// Mitsubishi GX Works2 project: BookEX6_17 Output   PLC: Q13UDV

// global labels: Global
VAR_GLOBAL
  bVar0 AT M5000 : BOOL;
  abArray0 AT M5010 : ARRAY [0..49] OF BOOL;
  sStr0 AT D5000 : STRING[199];
  sStr1 AT D5100 : STRING[199];
  sStr2 AT D5200 : STRING[199];
  sStr3 AT D5300 : STRING[199];
  sStr4 AT D5400 : STRING[199];
  sStr5 AT D5500 : STRING[199];
  sStr6 AT D5600 : STRING[199];
  sStr7 AT D5700 : STRING[199];
  sStr8 AT D5800 : STRING[199];
  sStr9 AT D5900 : STRING[199];
  iVar0 AT D4500 : INT;
  iVar1 AT D4501 : INT;
  iVar2 AT D4502 : INT;
  iVar3 AT D4503 : INT;
  iVar4 AT D4504 : INT;
  iVar5 AT D4505 : INT;
  iVar6 AT D4506 : INT;
  iVar7 AT D4507 : INT;
  iVar8 AT D4508 : INT;
  iVar9 AT D4509 : INT;
  dVar0 AT D4510 : DINT;
  dVar1 AT D4512 : DINT;
  dVar2 AT D4514 : DINT;
  dVar3 AT D4516 : DINT;
  dVar4 AT D4518 : DINT;
  dVar5 AT D4520 : DINT;
  dVar6 AT D4522 : DINT;
  dVar7 AT D4524 : DINT;
  dVar8 AT D4526 : DINT;
  dVar9 AT D4528 : DINT;
  wVar0 AT D4530 : WORD;
  wVar1 AT D4531 : WORD;
  wVar2 AT D4532 : WORD;
  wVar3 AT D4533 : WORD;
  wVar4 AT D4534 : WORD;
  wVar5 AT D4535 : WORD;
  wVar6 AT D4536 : WORD;
  wVar7 AT D4537 : WORD;
  wVar8 AT D4538 : WORD;
  wVar9 AT D4539 : WORD;
  dwVar0 AT D4540 : DWORD;
  dwVar1 AT D4542 : DWORD;
  dwVar2 AT D4544 : DWORD;
  dwVar3 AT D4546 : DWORD;
  dwVar4 AT D4548 : DWORD;
  dwVar5 AT D4550 : DWORD;
  dwVar6 AT D4552 : DWORD;
  dwVar7 AT D4554 : DWORD;
  dwVar8 AT D4556 : DWORD;
  dwVar9 AT D4558 : DWORD;
  fsVar0 AT D4560 : REAL;
  fsVar1 AT D4562 : REAL;
  fsVar2 AT D4564 : REAL;
  fsVar3 AT D4566 : REAL;
  fsVar4 AT D4568 : REAL;
  fsVar5 AT D4570 : REAL;
  fsVar6 AT D4572 : REAL;
  fsVar7 AT D4574 : REAL;
  fsVar8 AT D4576 : REAL;
  fsVar9 AT D4578 : REAL;
  fdVar0 AT D4580 : LREAL;
  tTime0 AT D4620 : TIME;
  tTime1 AT D4622 : TIME;
  tTime2 AT D4624 : TIME;
  tTime3 AT D4626 : TIME;
  tTime4 AT D4628 : TIME;
  tTime5 AT D4630 : TIME;
  tTime6 AT D4632 : TIME;
  tTime7 AT D4634 : TIME;
  tTime8 AT D4636 : TIME;
  tTime9 AT D4638 : TIME;
  tTime10 AT D4640 : TIME;
  bVar1 AT M5001 : BOOL;
  bVar2 AT M5002 : BOOL;
  bVar3 AT M5003 : BOOL;
  bVar4 AT M5004 : BOOL;
  bVar5 AT M5005 : BOOL;
  bVar6 AT M5006 : BOOL;
  bVar7 AT M5007 : BOOL;
  bVar8 AT M5008 : BOOL;
  bVar9 AT M5009 : BOOL;
  abArray1 AT M5060 : ARRAY [0..49] OF BOOL;
  abArray2 AT M5110 : ARRAY [0..49] OF BOOL;
  abArray3 AT M5160 : ARRAY [0..49] OF BOOL;
  abArray4 AT M5210 : ARRAY [0..49] OF BOOL;
  abArray5 AT M5260 : ARRAY [0..49] OF BOOL;
  abArray6 AT M5310 : ARRAY [0..49] OF BOOL;
  abArray7 AT M5360 : ARRAY [0..49] OF BOOL;
  abArray8 AT M5410 : ARRAY [0..49] OF BOOL;
  abArray9 AT M5460 : ARRAY [0..49] OF BOOL;
  fdVar1 AT D4584 : LREAL;
  fdVar2 AT D4588 : LREAL;
  fdVar3 AT D4592 : LREAL;
  fdVar4 AT D4596 : LREAL;
  fdVar5 AT D4600 : LREAL;
  fdVar6 AT D4604 : LREAL;
  fdVar7 AT D4608 : LREAL;
  fdVar8 AT D4612 : LREAL;
  fdVar9 AT D4616 : LREAL;
  aSendData1 AT D100 : ARRAY [0..9] OF INT;
  aiTxData AT D4000 : ARRAY [0..99] OF INT;
  aiRxData AT D4100 : ARRAY [0..99] OF INT;
  iOpenOK AT D3900 : INT;
  iOpenERR AT D3901 : INT;
  iSendOK AT D3902 : INT;
  iSendERR AT D3903 : INT;
  iCloseOK AT D3906 : INT;
  iCloseERR AT D3907 : INT;
  iRecvOK AT D3904 : INT;
  iRecvERR AT D3905 : INT;
  aiTxData2 AT D4200 : ARRAY [0..99] OF INT;
  aiRxData2 AT D4300 : ARRAY [0..99] OF INT;
  iOpenOK2 AT D3908 : INT;
  iOpenERR2 AT D3909 : INT;
  iSendOK2 AT D3910 : INT;
  iSendERR2 AT D3911 : INT;
  iRecvOK2 AT D3912 : INT;
  iRecvERR2 AT D3913 : INT;
  iCloseOK2 AT D3914 : INT;
  iCloseERR2 AT D3915 : INT;
  iEOpenComp AT D3916 : INT;
  iEOpenReq AT D3917 : INT;
  iERecvFlag AT D3918 : INT;
  iOpenCode AT D3919 : INT;
  iSendCode AT D3920 : INT;
  iRecvCode AT D3921 : INT;
  iCloseCode AT D3922 : INT;
  iOpenCode2 AT D3923 : INT;
  iSendCode2 AT D3924 : INT;
  iRecvCode2 AT D3925 : INT;
  iCloseCode2 AT D3926 : INT;
  aRecvData1 AT D110 : ARRAY [0..9] OF INT;
  aSendData2 AT D120 : ARRAY [0..9] OF INT;
  aRecvData2 AT D130 : ARRAY [0..9] OF INT;
END_VAR
// user libraries (not included): HMI

FUNCTION_BLOCK Flicker
VAR_INPUT
  t_Duty : TIME;
END_VAR
VAR_OUTPUT
  b_Lamp1 : BOOL;
  b_Lamp2 : BOOL;
END_VAR
VAR
  iInterval : INT;
END_VAR
;
iInterval := TIME_TO_INT(t_Duty) / 100;
OUT_T(NOT TS1, TC0, iInterval);
OUT_T(TS0, TC1, iInterval);
b_Lamp1 := TS0;
b_Lamp2 :=  NOT TS0;
END_FUNCTION_BLOCK

PROGRAM ExDELTA
VAR
  HMI05_1 : HMI05;
END_VAR
(* structured ladder/FBD written out as ST: instructions are called as NAME(EN, inputs, outputs); _pN, _eN, _tN stand for wires *)
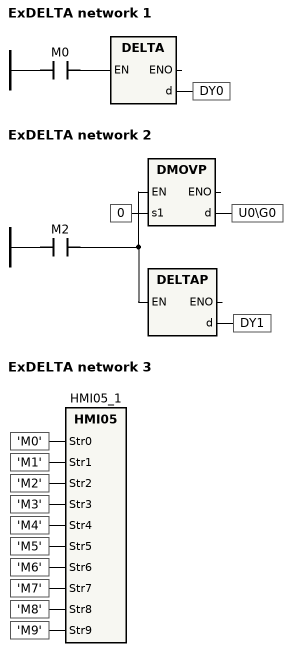
(* network 1 *)
DELTA(M0, DY0);
(* network 2 *)
DMOVP(M2, 0, U0\G0);
DELTAP(M2, DY1);
(* network 3 *)
HMI05_1(Str0 := 'M0', Str1 := 'M1', Str2 := 'M2', Str3 := 'M3', Str4 := 'M4', Str5 := 'M5', Str6 := 'M6', Str7 := 'M7', Str8 := 'M8', Str9 := 'M9');
END_PROGRAM

PROGRAM ExFF
VAR
  HMI05_1 : HMI05;
END_VAR
(* structured ladder/FBD written out as ST: instructions are called as NAME(EN, inputs, outputs); _pN, _eN, _tN stand for wires *)
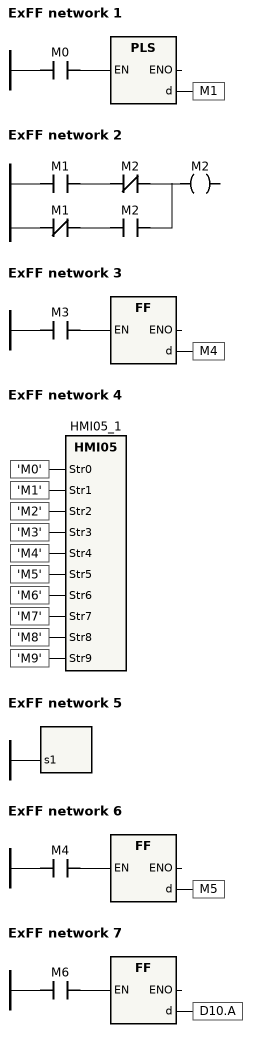
(* network 1 *)
PLS(M0, M1);
(* network 2 *)
M2 := (M1 AND NOT M2) OR (NOT M1 AND M2);
(* network 3 *)
FF(M3, M4);
(* network 4 *)
HMI05_1(Str0 := 'M0', Str1 := 'M1', Str2 := 'M2', Str3 := 'M3', Str4 := 'M4', Str5 := 'M5', Str6 := 'M6', Str7 := 'M7', Str8 := 'M8', Str9 := 'M9');
(* network 5 *)
(* element kind 10  <- TRUE *)
(* network 6 *)
FF(M4, M5);
(* network 7 *)
FF(M6, D10.A);
END_PROGRAM

PROGRAM ExFlicker
VAR
  HMI05_1 : HMI05;
  Flicker_1 : Flicker;
END_VAR
(* structured ladder/FBD written out as ST: instructions are called as NAME(EN, inputs, outputs); _pN, _eN, _tN stand for wires *)
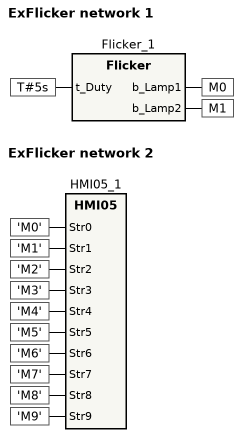
(* network 1 *)
Flicker_1(t_Duty := T#5s, b_Lamp1 => M0, b_Lamp2 => M1);
(* network 2 *)
HMI05_1(Str0 := 'M0', Str1 := 'M1', Str2 := 'M2', Str3 := 'M3', Str4 := 'M4', Str5 := 'M5', Str6 := 'M6', Str7 := 'M7', Str8 := 'M8', Str9 := 'M9');
END_PROGRAM

PROGRAM ExOUT
VAR
  HMI05_1 : HMI05;
END_VAR
(* structured ladder/FBD written out as ST: instructions are called as NAME(EN, inputs, outputs); _pN, _eN, _tN stand for wires *)
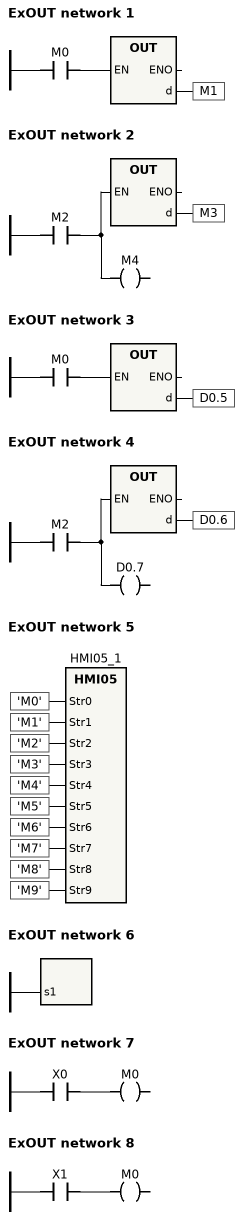
(* network 1 *)
OUT(M0, M1);
(* network 2 *)
OUT(M2, M3);
M4 := M2;
(* network 3 *)
OUT(M0, D0.5);
(* network 4 *)
OUT(M2, D0.6);
D0.7 := M2;
(* network 5 *)
HMI05_1(Str0 := 'M0', Str1 := 'M1', Str2 := 'M2', Str3 := 'M3', Str4 := 'M4', Str5 := 'M5', Str6 := 'M6', Str7 := 'M7', Str8 := 'M8', Str9 := 'M9');
(* network 6 *)
(* element kind 10  <- TRUE *)
(* network 7 *)
M0 := X0;
(* network 8 *)
M0 := X1;
END_PROGRAM

PROGRAM ExOut_C
VAR
  HMI05_1 : HMI05;
END_VAR
(* structured ladder/FBD written out as ST: instructions are called as NAME(EN, inputs, outputs); _pN, _eN, _tN stand for wires *)
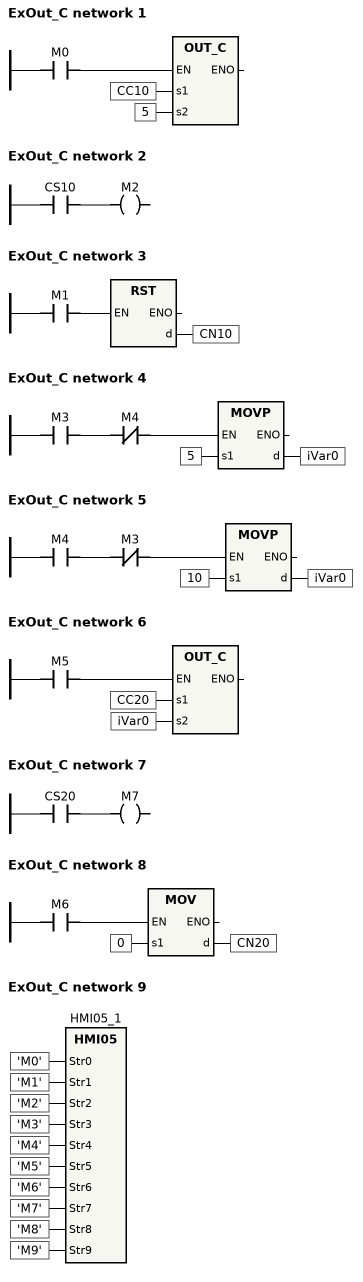
(* network 1 *)
OUT_C(M0, CC10, 5);
(* network 2 *)
M2 := CS10;
(* network 3 *)
RST(M1, CN10);
(* network 4 *)
MOVP(M3 AND NOT M4, 5, iVar0);
(* network 5 *)
MOVP(M4 AND NOT M3, 10, iVar0);
(* network 6 *)
OUT_C(M5, CC20, iVar0);
(* network 7 *)
M7 := CS20;
(* network 8 *)
MOV(M6, 0, CN20);
(* network 9 *)
HMI05_1(Str0 := 'M0', Str1 := 'M1', Str2 := 'M2', Str3 := 'M3', Str4 := 'M4', Str5 := 'M5', Str6 := 'M6', Str7 := 'M7', Str8 := 'M8', Str9 := 'M9');
END_PROGRAM

PROGRAM ExOut_T
VAR
  HMI05_1 : HMI05;
END_VAR
(* structured ladder/FBD written out as ST: instructions are called as NAME(EN, inputs, outputs); _pN, _eN, _tN stand for wires *)
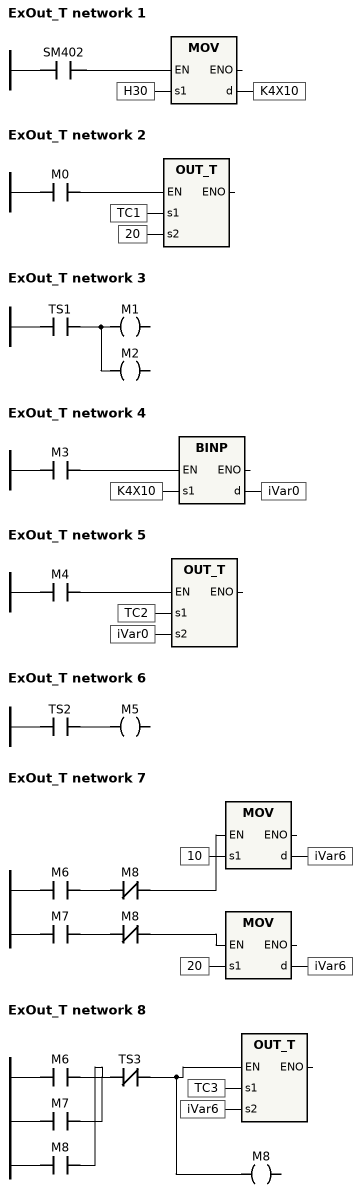
(* network 1 *)
MOV(SM402, H30, K4X10);
(* network 2 *)
OUT_T(M0, TC1, 20);
(* network 3 *)
M1 := TS1;
M2 := TS1;
(* network 4 *)
BINP(M3, K4X10, iVar0);
(* network 5 *)
OUT_T(M4, TC2, iVar0);
(* network 6 *)
M5 := TS2;
(* network 7 *)
MOV(M6 AND NOT M8, 10, iVar6);
MOV(M7 AND NOT M8, 20, iVar6);
(* network 8 *)
_p1 := (M6 OR M7 OR M8) AND NOT TS3;
M8 := _p1;
OUT_T(_p1, TC3, iVar6);
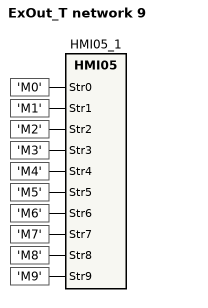
(* network 9 *)
HMI05_1(Str0 := 'M0', Str1 := 'M1', Str2 := 'M2', Str3 := 'M3', Str4 := 'M4', Str5 := 'M5', Str6 := 'M6', Str7 := 'M7', Str8 := 'M8', Str9 := 'M9');
END_PROGRAM

PROGRAM ExOut_T2
VAR
  HMI05_1 : HMI05;
END_VAR
(* structured ladder/FBD written out as ST: instructions are called as NAME(EN, inputs, outputs); _pN, _eN, _tN stand for wires *)
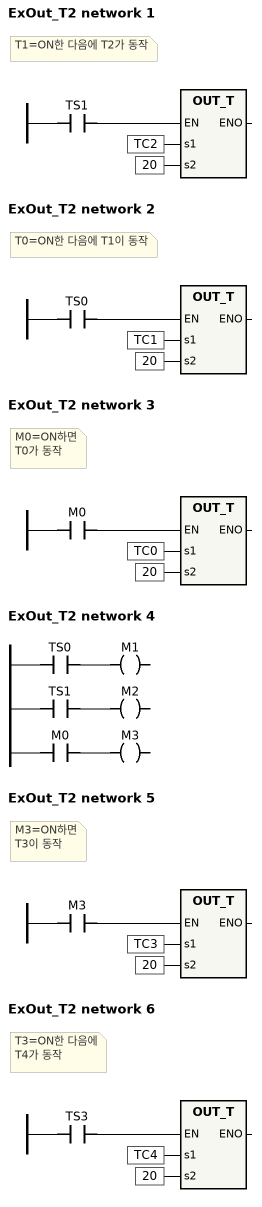
(* network 1 *)
(* T1=ON한 다음에 T2가 동작 *)
OUT_T(TS1, TC2, 20);
(* network 2 *)
(* T0=ON한 다음에 T1이 동작 *)
OUT_T(TS0, TC1, 20);
(* network 3 *)
(* M0=ON하면  / T0가 동작 *)
OUT_T(M0, TC0, 20);
(* network 4 *)
M1 := TS0;
M2 := TS1;
M3 := M0;
(* network 5 *)
(* M3=ON하면  / T3이 동작 *)
OUT_T(M3, TC3, 20);
(* network 6 *)
(* T3=ON한 다음에  / T4가 동작 *)
OUT_T(TS3, TC4, 20);
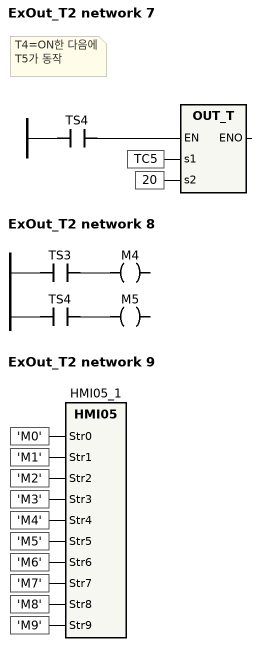
(* network 7 *)
(* T4=ON한 다음에  / T5가 동작 *)
OUT_T(TS4, TC5, 20);
(* network 8 *)
M4 := TS3;
M5 := TS4;
(* network 9 *)
HMI05_1(Str0 := 'M0', Str1 := 'M1', Str2 := 'M2', Str3 := 'M3', Str4 := 'M4', Str5 := 'M5', Str6 := 'M6', Str7 := 'M7', Str8 := 'M8', Str9 := 'M9');
END_PROGRAM

PROGRAM ExPLF
VAR
  HMI05_1 : HMI05;
END_VAR
(* structured ladder/FBD written out as ST: instructions are called as NAME(EN, inputs, outputs); _pN, _eN, _tN stand for wires *)
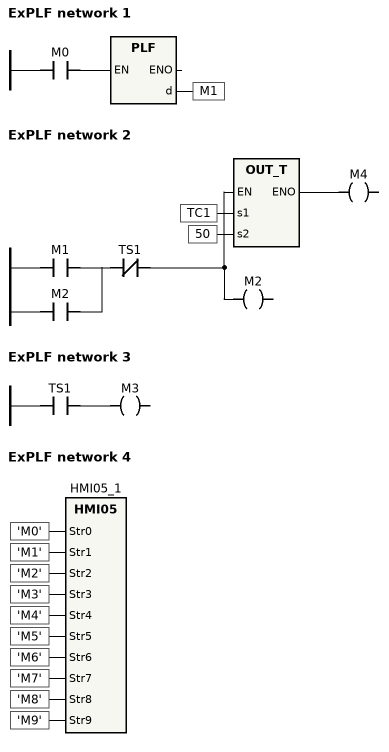
(* network 1 *)
PLF(M0, M1);
(* network 2 *)
_p1 := (M1 OR M2) AND NOT TS1;
_e2 := OUT_T(_p1, TC1, 50);
M4 := _e2;
M2 := _p1;
(* network 3 *)
M3 := TS1;
(* network 4 *)
HMI05_1(Str0 := 'M0', Str1 := 'M1', Str2 := 'M2', Str3 := 'M3', Str4 := 'M4', Str5 := 'M5', Str6 := 'M6', Str7 := 'M7', Str8 := 'M8', Str9 := 'M9');
END_PROGRAM

PROGRAM ExPLS
VAR
  HMI05_1 : HMI05;
END_VAR
(* structured ladder/FBD written out as ST: instructions are called as NAME(EN, inputs, outputs); _pN, _eN, _tN stand for wires *)
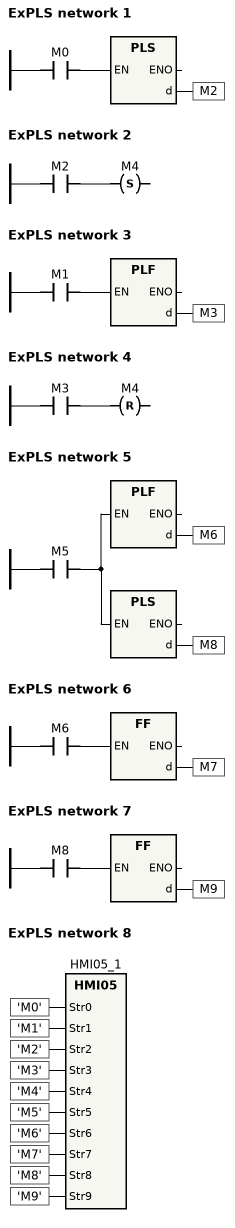
(* network 1 *)
PLS(M0, M2);
(* network 2 *)
SET(M2, M4);
(* network 3 *)
PLF(M1, M3);
(* network 4 *)
RST(M3, M4);
(* network 5 *)
PLF(M5, M6);
PLS(M5, M8);
(* network 6 *)
FF(M6, M7);
(* network 7 *)
FF(M8, M9);
(* network 8 *)
HMI05_1(Str0 := 'M0', Str1 := 'M1', Str2 := 'M2', Str3 := 'M3', Str4 := 'M4', Str5 := 'M5', Str6 := 'M6', Str7 := 'M7', Str8 := 'M8', Str9 := 'M9');
END_PROGRAM

PROGRAM ExPowerOn
VAR
  bPowerFail : BOOL;
  TON_1 : TON;
  TON_2 : TON;
  bOff : BOOL;
  bOn : BOOL;
  TON_3 : TON;
  HMI05_1 : HMI05;
END_VAR
(* structured ladder/FBD written out as ST: instructions are called as NAME(EN, inputs, outputs); _pN, _eN, _tN stand for wires *)
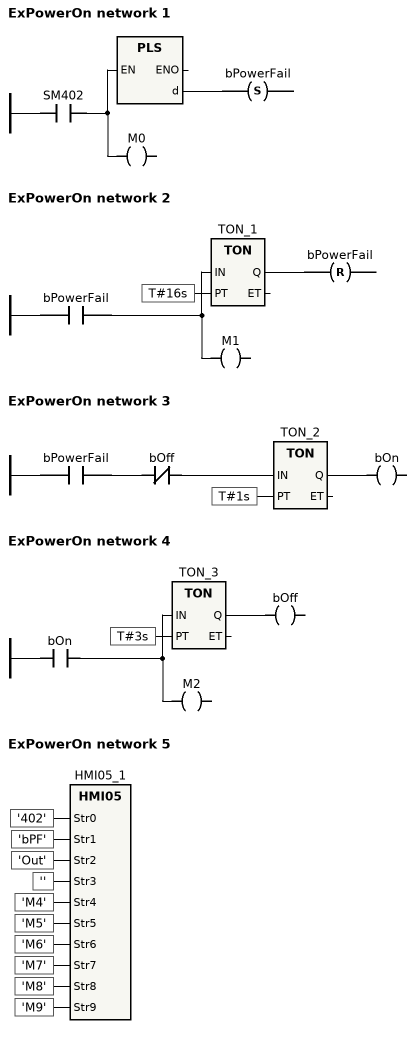
(* network 1 *)
PLS(SM402, _t1);
SET(_t1, bPowerFail);
M0 := SM402;
(* network 2 *)
TON_1(IN := bPowerFail, PT := T#16s);
RST(TON_1.Q, bPowerFail);
M1 := bPowerFail;
(* network 3 *)
TON_2(IN := bPowerFail AND NOT bOff, PT := T#1s);
bOn := TON_2.Q;
(* network 4 *)
TON_3(IN := bOn, PT := T#3s);
bOff := TON_3.Q;
M2 := bOn;
(* network 5 *)
HMI05_1(Str0 := '402', Str1 := 'bPF', Str2 := 'Out', Str3 := '', Str4 := 'M4', Str5 := 'M5', Str6 := 'M6', Str7 := 'M7', Str8 := 'M8', Str9 := 'M9');
END_PROGRAM

PROGRAM ExPowerOn2
VAR
  bPowerFail : BOOL;
  TON_1 : TON;
  TON_2 : TON;
  bOff : BOOL;
  bOn : BOOL;
  TON_3 : TON;
  HMI05_1 : HMI05;
END_VAR
(* structured ladder/FBD written out as ST: instructions are called as NAME(EN, inputs, outputs); _pN, _eN, _tN stand for wires *)
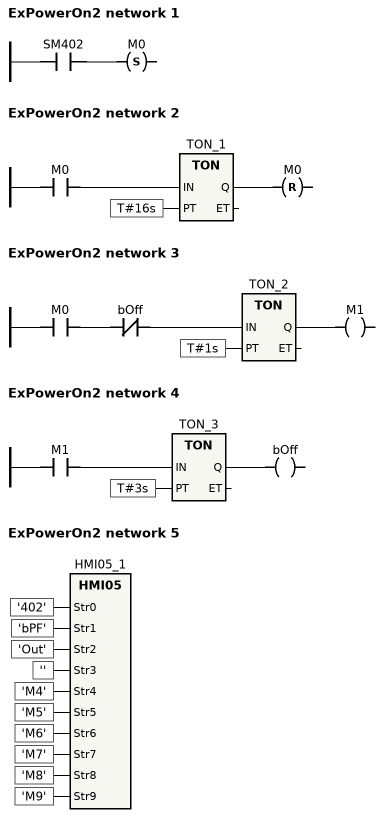
(* network 1 *)
SET(SM402, M0);
(* network 2 *)
TON_1(IN := M0, PT := T#16s);
RST(TON_1.Q, M0);
(* network 3 *)
TON_2(IN := M0 AND NOT bOff, PT := T#1s);
M1 := TON_2.Q;
(* network 4 *)
TON_3(IN := M1, PT := T#3s);
bOff := TON_3.Q;
(* network 5 *)
HMI05_1(Str0 := '402', Str1 := 'bPF', Str2 := 'Out', Str3 := '', Str4 := 'M4', Str5 := 'M5', Str6 := 'M6', Str7 := 'M7', Str8 := 'M8', Str9 := 'M9');
END_PROGRAM

PROGRAM ExSET
VAR
  HMI05_1 : HMI05;
END_VAR
(* structured ladder/FBD written out as ST: instructions are called as NAME(EN, inputs, outputs); _pN, _eN, _tN stand for wires *)
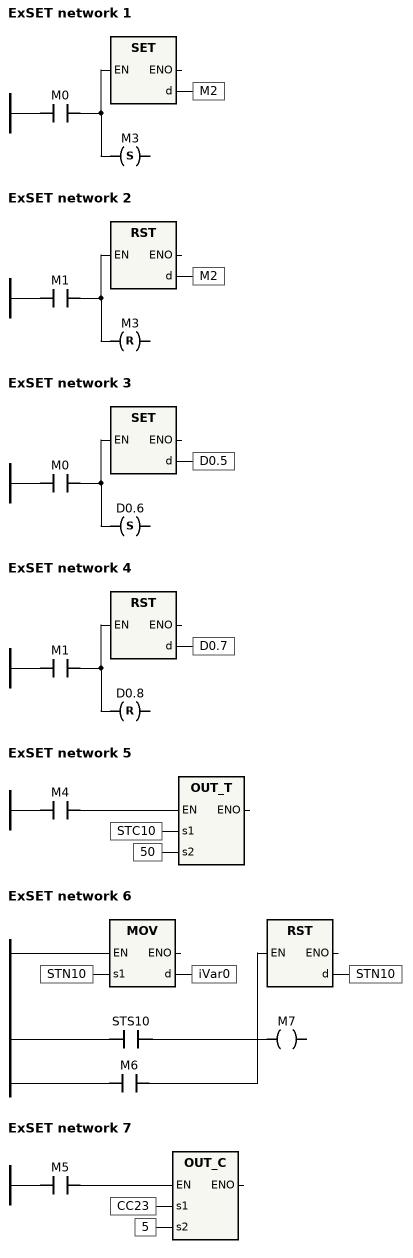
(* network 1 *)
SET(M0, M2);
SET(M0, M3);
(* network 2 *)
RST(M1, M2);
RST(M1, M3);
(* network 3 *)
SET(M0, D0.5);
SET(M0, D0.6);
(* network 4 *)
RST(M1, D0.7);
RST(M1, D0.8);
(* network 5 *)
OUT_T(M4, STC10, 50);
(* network 6 *)
M7 := STS10;
MOV(TRUE, STN10, iVar0);
RST(M6, STN10);
(* network 7 *)
OUT_C(M5, CC23, 5);
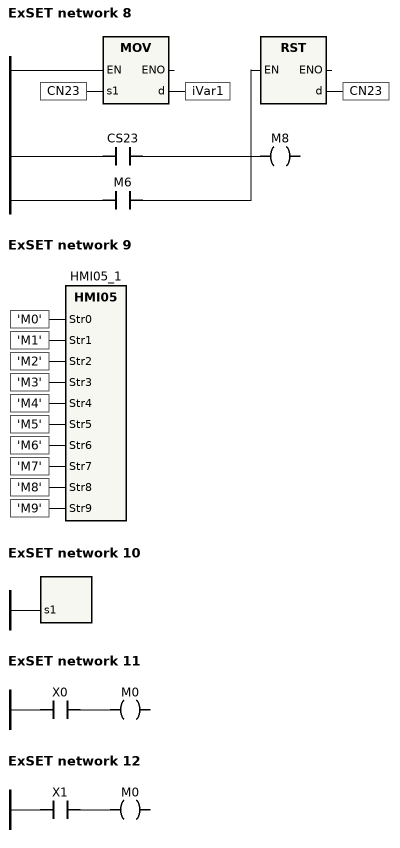
(* network 8 *)
M8 := CS23;
MOV(TRUE, CN23, iVar1);
RST(M6, CN23);
(* network 9 *)
HMI05_1(Str0 := 'M0', Str1 := 'M1', Str2 := 'M2', Str3 := 'M3', Str4 := 'M4', Str5 := 'M5', Str6 := 'M6', Str7 := 'M7', Str8 := 'M8', Str9 := 'M9');
(* network 10 *)
(* element kind 10  <- TRUE *)
(* network 11 *)
M0 := X0;
(* network 12 *)
M0 := X1;
END_PROGRAM

PROGRAM ExFF3
VAR
  HMI05_1 : HMI05;
END_VAR
(* structured ladder/FBD written out as ST: instructions are called as NAME(EN, inputs, outputs); _pN, _eN, _tN stand for wires *)
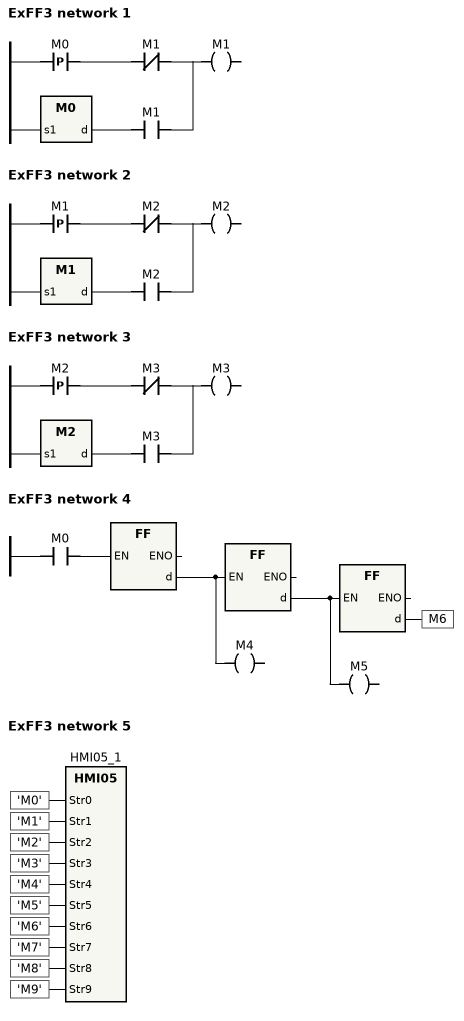
(* network 1 *)
(* element kind 19 M0 <- TRUE *)
M1 := (LDP(TRUE, M0) AND NOT M1) OR (_feedback AND M1);
(* network 2 *)
(* element kind 19 M1 <- TRUE *)
M2 := (LDP(TRUE, M1) AND NOT M2) OR (_feedback AND M2);
(* network 3 *)
(* element kind 19 M2 <- TRUE *)
M3 := (LDP(TRUE, M2) AND NOT M3) OR (_feedback AND M3);
(* network 4 *)
FF(M0, _t1);
FF(_t1, _t2);
FF(_t2, M6);
M4 := _t1;
M5 := _t2;
(* network 5 *)
HMI05_1(Str0 := 'M0', Str1 := 'M1', Str2 := 'M2', Str3 := 'M3', Str4 := 'M4', Str5 := 'M5', Str6 := 'M6', Str7 := 'M7', Str8 := 'M8', Str9 := 'M9');
END_PROGRAM

PROGRAM ExFF2
VAR
  HMI05_1 : HMI05;
END_VAR
(* structured ladder/FBD written out as ST: instructions are called as NAME(EN, inputs, outputs); _pN, _eN, _tN stand for wires *)
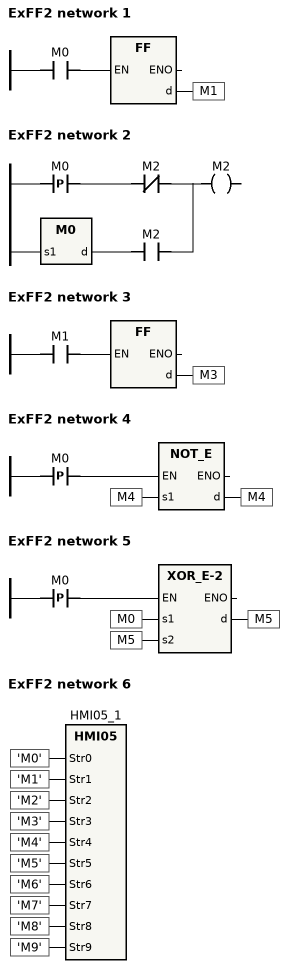
(* network 1 *)
FF(M0, M1);
(* network 2 *)
(* element kind 19 M0 <- TRUE *)
M2 := (LDP(TRUE, M0) AND NOT M2) OR (_feedback AND M2);
(* network 3 *)
FF(M1, M3);
(* network 4 *)
NOT_E(LDP(TRUE, M0), M4, M4);
(* network 5 *)
XOR_E(LDP(TRUE, M0), M0, M5, M5);
(* network 6 *)
HMI05_1(Str0 := 'M0', Str1 := 'M1', Str2 := 'M2', Str3 := 'M3', Str4 := 'M4', Str5 := 'M5', Str6 := 'M6', Str7 := 'M7', Str8 := 'M8', Str9 := 'M9');
END_PROGRAM

PROGRAM ExPLS2
VAR
  HMI05_1 : HMI05;
END_VAR
(* structured ladder/FBD written out as ST: instructions are called as NAME(EN, inputs, outputs); _pN, _eN, _tN stand for wires *)
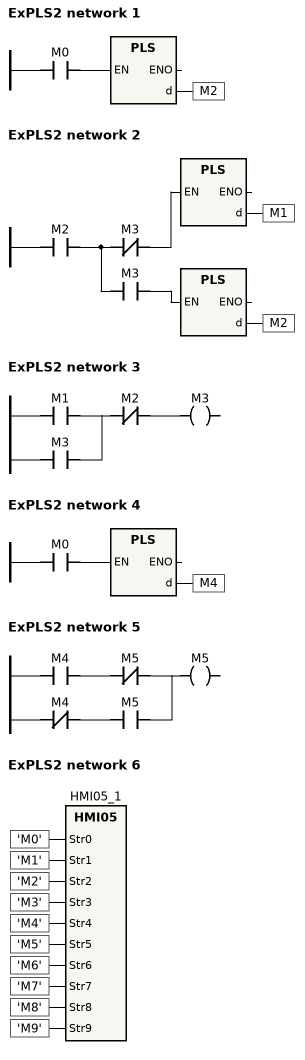
(* network 1 *)
PLS(M0, M2);
(* network 2 *)
PLS(M2 AND NOT M3, M1);
PLS(M2 AND M3, M2);
(* network 3 *)
M3 := (M1 OR M3) AND NOT M2;
(* network 4 *)
PLS(M0, M4);
(* network 5 *)
M5 := (M4 AND NOT M5) OR (NOT M4 AND M5);
(* network 6 *)
HMI05_1(Str0 := 'M0', Str1 := 'M1', Str2 := 'M2', Str3 := 'M3', Str4 := 'M4', Str5 := 'M5', Str6 := 'M6', Str7 := 'M7', Str8 := 'M8', Str9 := 'M9');
END_PROGRAM

PROGRAM ExOut_T_C
VAR
  HMI20_1 : HMI20;
  Mov8INT_1 : Mov8INT;
END_VAR
(* structured ladder/FBD written out as ST: instructions are called as NAME(EN, inputs, outputs); _pN, _eN, _tN stand for wires *)
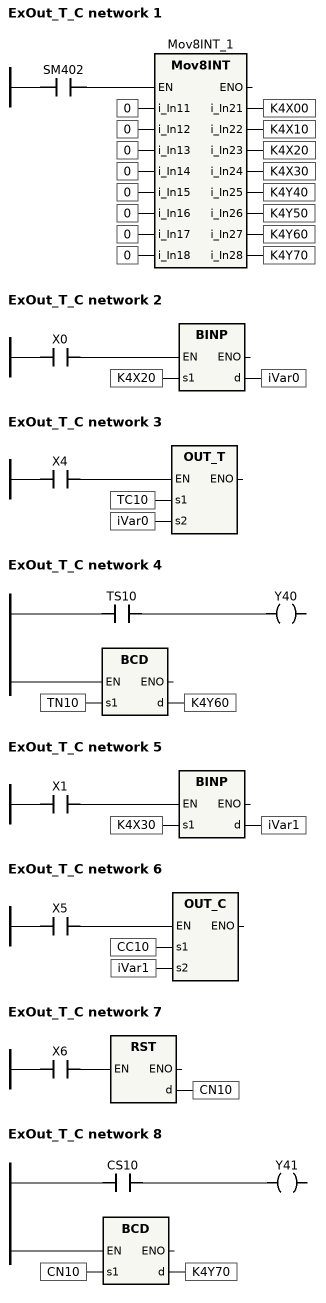
(* network 1 *)
Mov8INT_1(EN := SM402, i_In11 := 0, i_In12 := 0, i_In13 := 0, i_In14 := 0, i_In15 := 0, i_In16 := 0, i_In17 := 0, i_In18 := 0, i_In21 => K4X00, i_In22 => K4X10, i_In23 => K4X20, i_In24 => K4X30, i_In25 => K4Y40, i_In26 => K4Y50, i_In27 => K4Y60, i_In28 => K4Y70);
(* network 2 *)
BINP(X0, K4X20, iVar0);
(* network 3 *)
OUT_T(X4, TC10, iVar0);
(* network 4 *)
Y40 := TS10;
BCD(TRUE, TN10, K4Y60);
(* network 5 *)
BINP(X1, K4X30, iVar1);
(* network 6 *)
OUT_C(X5, CC10, iVar1);
(* network 7 *)
RST(X6, CN10);
(* network 8 *)
Y41 := CS10;
BCD(TRUE, CN10, K4Y70);
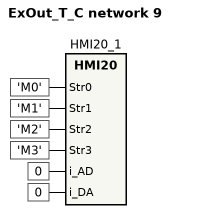
(* network 9 *)
HMI20_1(Str0 := 'M0', Str1 := 'M1', Str2 := 'M2', Str3 := 'M3', i_AD := 0, i_DA := 0);
END_PROGRAM

PROGRAM ExXOR
VAR
  HMI05_1 : HMI05;
  bOutput0 : BOOL;
  bOutput1 : BOOL;
END_VAR
(* structured ladder/FBD written out as ST: instructions are called as NAME(EN, inputs, outputs); _pN, _eN, _tN stand for wires *)
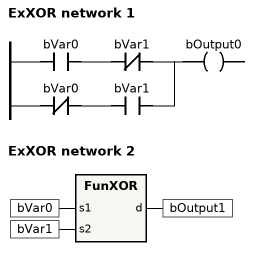
(* network 1 *)
bOutput0 := (bVar0 AND NOT bVar1) OR (NOT bVar0 AND bVar1);
(* network 2 *)
bOutput1 := FunXOR(bVar0, bVar1);
END_PROGRAM

FUNCTION FunXOR
VAR_INPUT
  Var0 : BOOL;
  Var1 : BOOL;
END_VAR
;

FunXOR := Var0 XOR Var1;
END_FUNCTION
